FUNCTION_BLOCK FB_T_FF (* Toggle flip-flop on clock edge *)
  (* Standard: 61499-1; Description: Copyright (c) 2023 Martin Erich Jobst This program and the accompanying materials are made available under the terms of the Eclipse Public License 2.0 which is available at https://www.eclipse.org/legal/epl-2.0/ SPDX-License-Identifier: EPL-2.0 *)
  (* Version 3.0, 2025-04-14, Patrick Aigner, changed package *)
  (* Version 1.0, 2023-04-28, Martin Jobst *)
  PACKAGE logiBUS::bistableElements;
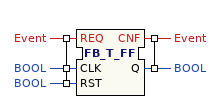
  EVENT_INPUT
    REQ WITH CLK, RST; (* Normal Execution Request *)
  END_EVENT
  EVENT_OUTPUT
    CNF WITH Q; (* Execution Confirmation *)
  END_EVENT
  VAR_INPUT
    CLK : BOOL; (* Clock *)
    RST : BOOL; (* Reset *)
  END_VAR
  VAR_OUTPUT
    Q : BOOL; (* Output *)
  END_VAR
  VAR
    EDGE : BOOL := TRUE;
  END_VAR
  EC_STATES
    REQ : REQ -> CNF;
  END_STATES
  ALGORITHM REQ IN ST:
IF RST THEN
	Q := BOOL#FALSE;
ELSIF CLK AND NOT EDGE THEN
	Q := NOT Q;
END_IF;
EDGE := CLK;
  END_ALGORITHM
END_FUNCTION_BLOCK
